// TIA Portal V17 export
// export: Created 2024-09-02T12:49:56.9664933Z, ExportSetting WithDefaults, DisplayName Totally Integrated Automation Portal, DisplayVersion V17, DisplayName TIA Portal Openness, DisplayVersion V17, DisplayName TIA Portal Version Control Interface, DisplayVersion V17, DisplayName STEP 7 Professional, DisplayVersion V17, DisplayName STEP 7 Safety, DisplayVersion V17, DisplayName WinCC Professional, DisplayVersion V17
FUNCTION_BLOCK "AnwFB_CycleTimes"   // FB1992, LAD
{ S7_Optimized_Access := 'TRUE' }
VERSION : 0.1
// stored: AutoNumber false, IsIECCheckEnabled false, IsRetainMemResEnabled false, MemoryReserve 100, SetENOAutomatically false, UDAEnableTagReadback false
   VAR_INPUT
      Start : Bool;
      Break : Bool;
      Stop : Bool;
      Precission : Int := 10;
   END_VAR
   VAR_OUTPUT
      CycleTimeExceeded : Bool;
   END_VAR
   VAR_IN_OUT
      CycleTimeIndex : Int;
      MainScreenField : DInt;
      dataDB : "LTLL_typeData";
      configDB : "LTLL_typeConfig";
   END_VAR
   VAR
      FP : Array[1..16] of Bool;
      StartTime : Time;
      StartBreakTime : Time;
      StopBreakTime : Time;
      CurrentBreak : Time;
      TotalBreak : Time;
      StopTime : Time;
      CycleTime : Time;
      DIntCycleTime : DWord;
      IntCycleTime : Byte;
      sPrecission : Int;
   END_VAR
   VAR_TEMP
      tBreakCalcEnd : Bool;
      tCycleTimeEnd : Bool;
   END_VAR
   VAR_TEMP   // added for the SCL form of the ladder/FBD networks
      _w1 : Bool;
      _w2 : Bool;
      _w3 : Bool;
   END_VAR
BEGIN

REGION Network 1: Init Precission
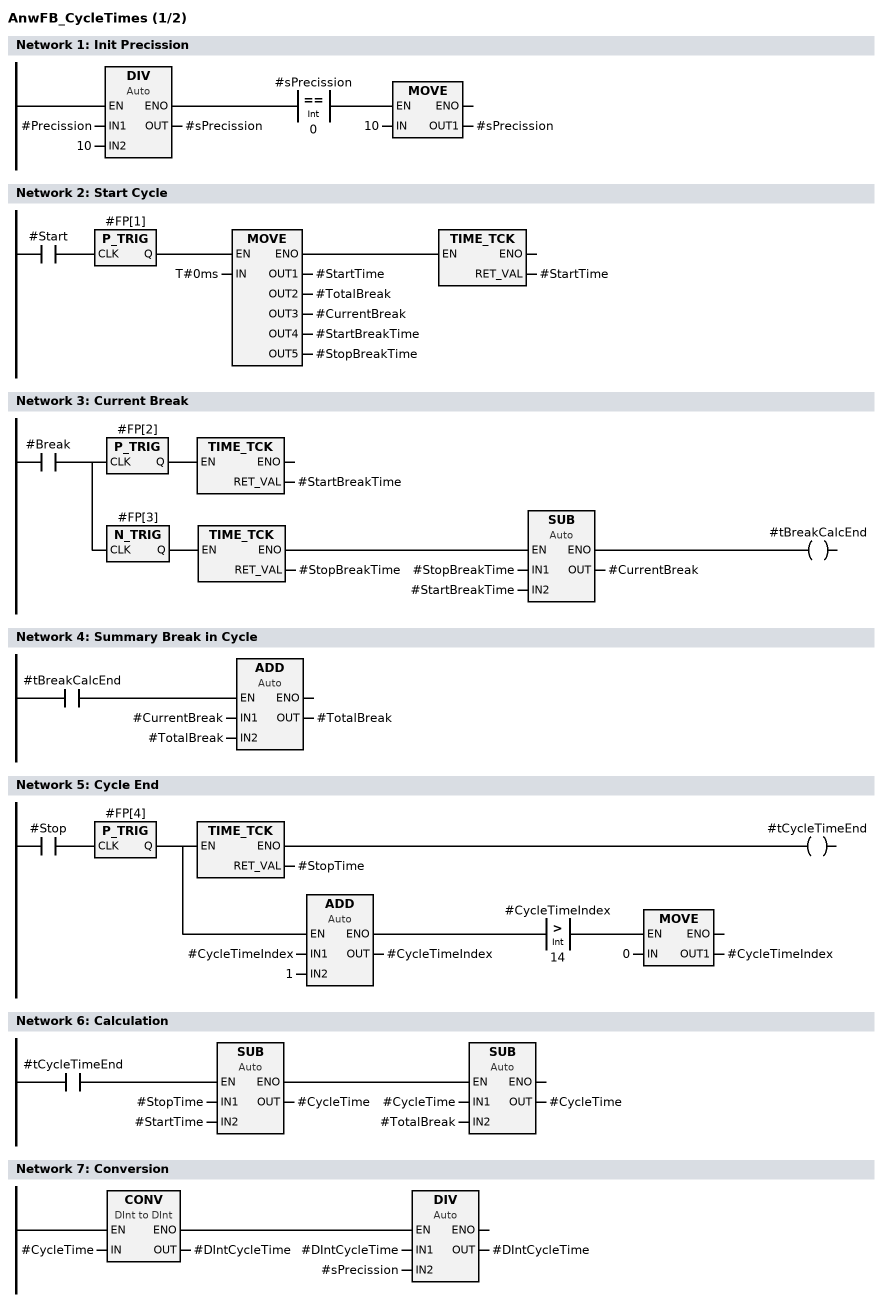
   RUNG wire#powerrail
      Div(in1 := #Precission, in2 := 10, out => #sPrecission)
      { S7_Templates := "SrcType := Int" } EQ_Contact(in1 := #sPrecission, in2 := 0)
      Move(in := 10, out1 => #sPrecission)
   END_RUNG
   // the same network as SCL:
   #sPrecission := #Precission / 10;
   IF #sPrecission = 0 THEN #sPrecission := 10; END_IF;
END_REGION

REGION Network 2: Start Cycle
   RUNG wire#powerrail
      Contact( #Start )
      P_Trig( #FP[1] )
      Move(in := T#0ms, out1 => #StartTime, out2 => #TotalBreak, out3 => #CurrentBreak, out4 => #StartBreakTime, out5 => #StopBreakTime)
      TIME_TCK(RET_VAL => #StartTime)
   END_RUNG
   // the same network as SCL:
   #_w1 := #Start AND NOT #FP[1];   // rising edge
   #FP[1] := #Start;
   IF #_w1 THEN
       #StartTime := T#0ms;
       #TotalBreak := T#0ms;
       #CurrentBreak := T#0ms;
       #StartBreakTime := T#0ms;
       #StopBreakTime := T#0ms;
       #StartTime := TIME_TCK();
   END_IF;
END_REGION

REGION Network 3: Current Break
   RUNG wire#powerrail
      Contact( #Break )
      wire#w1
      P_Trig( #FP[2] )
      TIME_TCK(RET_VAL => #StartBreakTime)
   END_RUNG
   RUNG wire#w1
      N_Trig( #FP[3] )
      TIME_TCK(RET_VAL => #StopBreakTime)
      Sub(in1 := #StopBreakTime, in2 := #StartBreakTime, out => #CurrentBreak)
      Coil( #tBreakCalcEnd )
   END_RUNG
   // the same network as SCL:
   #_w1 := #Break AND NOT #FP[2];   // rising edge
   #FP[2] := #Break;
   IF #_w1 THEN #StartBreakTime := TIME_TCK(); END_IF;
   #_w2 := NOT #Break AND #FP[3];   // falling edge
   #FP[3] := #Break;
   #StopBreakTime := TIME_TCK(EN := #_w2, ENO => #_w3);
   IF #_w3 THEN #CurrentBreak := #StopBreakTime - #StartBreakTime; END_IF;
   #tBreakCalcEnd := #_w3;
END_REGION

REGION Network 4: Summary Break in Cycle
   RUNG wire#powerrail
      Contact( #tBreakCalcEnd )
      Add(in1 := #CurrentBreak, in2 := #TotalBreak, out => #TotalBreak)
   END_RUNG
   // the same network as SCL:
   IF #tBreakCalcEnd THEN #TotalBreak := #CurrentBreak + #TotalBreak; END_IF;
END_REGION

REGION Network 5: Cycle End
   RUNG wire#powerrail
      Contact( #Stop )
      P_Trig( #FP[4] )
      wire#w1
      TIME_TCK(RET_VAL => #StopTime)
      Coil( #tCycleTimeEnd )
   END_RUNG
   RUNG wire#w1
      Add(in1 := #CycleTimeIndex, in2 := 1, out => #CycleTimeIndex)
      { S7_Templates := "SrcType := Int" } GT_Contact(in1 := #CycleTimeIndex, in2 := 14)
      Move(in := 0, out1 => #CycleTimeIndex)
   END_RUNG
   // the same network as SCL:
   #_w1 := #Stop AND NOT #FP[4];   // rising edge
   #FP[4] := #Stop;
   #StopTime := TIME_TCK(EN := #_w1, ENO => #_w2);
   #tCycleTimeEnd := #_w2;
   IF #_w1 THEN #CycleTimeIndex := #CycleTimeIndex + 1; END_IF;
   IF #_w1 AND (#CycleTimeIndex > 14) THEN #CycleTimeIndex := 0; END_IF;
END_REGION

REGION Network 6: Calculation
   RUNG wire#powerrail
      Contact( #tCycleTimeEnd )
      Sub(in1 := #StopTime, in2 := #StartTime, out => #CycleTime)
      Sub(in1 := #CycleTime, in2 := #TotalBreak, out => #CycleTime)
   END_RUNG
   // the same network as SCL:
   IF #tCycleTimeEnd THEN
       #CycleTime := #StopTime - #StartTime;
       #CycleTime := #CycleTime - #TotalBreak;
   END_IF;
END_REGION

REGION Network 7: Conversion
   RUNG wire#powerrail
      { S7_Templates := "[SrcType := DInt, DestType := DInt]" } Convert(in := #CycleTime, out => #DIntCycleTime)
      Div(in1 := #DIntCycleTime, in2 := #sPrecission, out => #DIntCycleTime)
   END_RUNG
   // the same network as SCL:
   #DIntCycleTime := DINT_TO_DINT(#CycleTime);
   #DIntCycleTime := #DIntCycleTime / #sPrecission;
END_REGION

REGION Network 8: Save Data to Wright Data Area in LTLL_Data
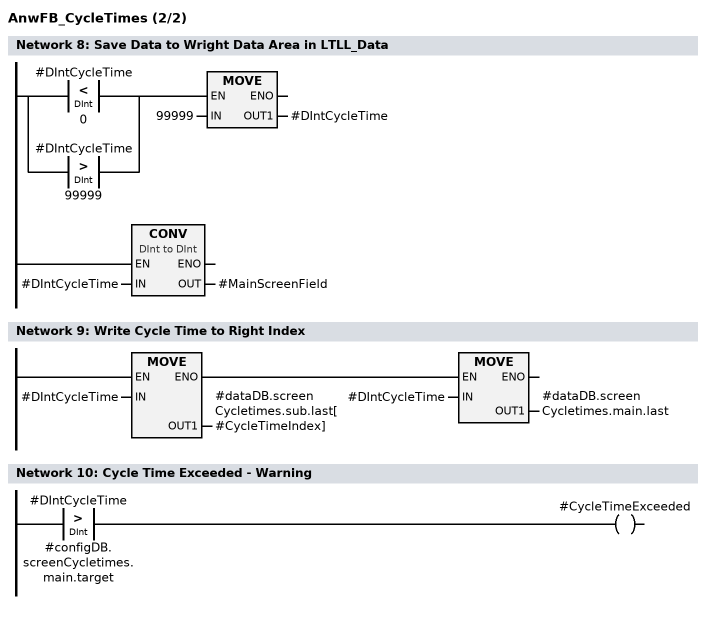
   RUNG wire#powerrail
      { S7_Templates := "SrcType := DInt" } LT_Contact(in1 := #DIntCycleTime, in2 := 0)
      wire#w1
      Move(in := 99999, out1 => #DIntCycleTime)
   END_RUNG
   RUNG wire#powerrail
      { S7_Templates := "SrcType := DInt" } GT_Contact(in1 := #DIntCycleTime, in2 := 99999)
   END_RUNG wire#w1
   RUNG wire#powerrail
      { S7_Templates := "[SrcType := DInt, DestType := DInt]" } Convert(in := #DIntCycleTime, out => #MainScreenField)
   END_RUNG
   // the same network as SCL:
   IF (#DIntCycleTime < 0) OR (#DIntCycleTime > 99999) THEN #DIntCycleTime := 99999; END_IF;
   #MainScreenField := DINT_TO_DINT(#DIntCycleTime);
END_REGION

REGION Network 9: Write Cycle Time to Right Index
   RUNG wire#powerrail
      Move(in := #DIntCycleTime, out1 => #dataDB.screenCycletimes.sub.last[#CycleTimeIndex])
      Move(in := #DIntCycleTime, out1 => #dataDB.screenCycletimes.main.last)
   END_RUNG
   // the same network as SCL:
   #dataDB.screenCycletimes.sub.last[#CycleTimeIndex] := #DIntCycleTime;
   #dataDB.screenCycletimes.main.last := #DIntCycleTime;
END_REGION

REGION Network 10: Cycle Time Exceeded - Warning
   RUNG wire#powerrail
      { S7_Templates := "SrcType := DInt" } GT_Contact(in1 := #DIntCycleTime, in2 := #configDB.screenCycletimes.main.target)
      Coil( #CycleTimeExceeded )
   END_RUNG
   // the same network as SCL:
   #CycleTimeExceeded := #DIntCycleTime > #configDB.screenCycletimes.main.target;
END_REGION
END_FUNCTION_BLOCK
